// TIA Portal V17 export
// export: Created 2022-07-28T18:02:49.2416431Z, ExportSetting None, DisplayName Totally Integrated Automation Portal, DisplayVersion V17, DisplayName TIA Portal Openness, DisplayVersion V17, DisplayName TIA Portal Teamcenter Gateway, DisplayVersion V17, DisplayName TIA Portal Version Control Interface, DisplayVersion V17, DisplayName TIA Portal Test Suite Advanced, DisplayVersion V17, DisplayName SINAMICS Startdrive Advanced, DisplayVersion V17, DisplayName SINAMICS DCC, DisplayVersion V17, DisplayName SINAMICS Startdrive G130, G150, S120, S150, SINAMICS MV, S210, DisplayVersion V17, DisplayName SINAMICS Startdrive G110M, G120, G120C, G120D, G120P, G115D, DisplayVersion V17, DisplayName STEP 7 Professional, DisplayVersion V17, DisplayName SIMATIC Energy Suite, DisplayVersion V17, DisplayName STEP 7 CFC, DisplayVersion V17, DisplayName STEP 7 Safety, DisplayVersion V17, DisplayName WinCC Advanced / Unified PC, DisplayVersion V17, DisplayName SIMATIC Visualization Architect, DisplayVersion V17
FUNCTION "Lib_FC_PID_Cascad_SortPrior" : "_PID_Cascad_AutoCtrlPumpsAll"   // FC22, SCL
{ S7_Optimized_Access := 'TRUE' }
// stored: SetENOAutomatically false
   VAR_INPUT
      i_InputArr : "_PID_Cascad_AutoCtrlPumpsAll";
   END_VAR
   VAR_TEMP
      ti_MinPrior : Int;
      ti_CntOut : Int;
      ti_CntIn : Int;
      ti_NMinPrior : Int;
      t_TempOnePump : "_PID_Cascad_AutoCtrlPumpsOne";
   END_VAR
BEGIN
   #Lib_FC_PID_Cascad_SortPrior := #i_InputArr;

   //Go loop for find min prior
   FOR #ti_CntOut := 0 TO 2 DO
       #ti_MinPrior := #Lib_FC_PID_Cascad_SortPrior.Arr[#ti_CntOut].i_Priority;
       #ti_NMinPrior := #ti_CntOut;

       //Go for find min prior
       FOR #ti_CntIn := #ti_CntOut TO 2 DO
           IF #ti_MinPrior > #Lib_FC_PID_Cascad_SortPrior.Arr[#ti_CntIn].i_Priority
           THEN
               #ti_MinPrior := #Lib_FC_PID_Cascad_SortPrior.Arr[#ti_CntIn].i_Priority;
               #ti_NMinPrior := #ti_CntIn;
           END_IF;
       END_FOR;

       //Asign min priority
       #t_TempOnePump := #Lib_FC_PID_Cascad_SortPrior.Arr[#ti_CntOut];
       #Lib_FC_PID_Cascad_SortPrior.Arr[#ti_CntOut] := #Lib_FC_PID_Cascad_SortPrior.Arr[#ti_NMinPrior];
       #Lib_FC_PID_Cascad_SortPrior.Arr[#ti_NMinPrior] := #t_TempOnePump;
   END_FOR;
END_FUNCTION
